VAR_GLOBAL CONSTANT
	MAX_QUEUE_SIZE : INT:= 10;

END_VAR

(* stored: Version 1.1.0.1, ProductVersion 3.1.4018.5
   GVL Param_Queue: Id {5aa83e05-0926-46b4-b14e-d5fed114d936}, ParameterList True *)
